// TwinCAT 3 PLC project HeatPumpTestBenchControl
// ProgramVersion: 3.1.4022.1
// CompilerDefines: VISU_USEPROPERTYINFO
// libraries:
//   Tc2_ControllerToolbox, * (Beckhoff Automation GmbH)
//   Tc2_Standard, * (Beckhoff Automation GmbH)
//   Tc2_System, * (Beckhoff Automation GmbH)
//   Tc2_TempController, * (Beckhoff Automation GmbH)
//   Tc2_Utilities, * (Beckhoff Automation GmbH)
//   Tc3_Module, * (Beckhoff Automation GmbH)
//   VisuDialogs, * (System)
// project tree:
//   DUTs/ E_PowMeas.TcDUT (not stored), E_Press.TcDUT (not stored), E_TempSensVR10.TcDUT (not stored), E_TempSensPT100.TcDUT (not stored), E_IndexPowMeas.TcDUT (not stored), E_SMStatus.TcDUT (not stored), E_TempSensVR11.TcDUT (not stored), E_Terminals.TcDUT (not stored), ST_InputVar.TcDUT (not stored), ST_InputVar_PowMeas.TcDUT (not stored), ST_OutputVar.TcDUT (not stored), ST_PumpTime.TcDUT (not stored)
//   / GlobalTextList.TcGTLO (not stored), PlcTask.TcTTO (not stored), Visualization Manager.TcVMO (not stored)
//   GVLs/ DigOutputs.TcGVL (not stored), HeatingCurve.TcGVL (not stored), AnaOutputs.TcGVL (not stored), PID.TcGVL (not stored), PowMeas.TcGVL (not stored), Pressures.TcGVL (not stored), PumpTiming.TcGVL (not stored), StateMachine.TcGVL (not stored), SysCheck.TcGVL (not stored), SysCheckParams.TcGVL (not stored), TempConvDat.TcGVL (not stored), Temperatures.TcGVL (not stored), TempSetpoints.TcGVL (not stored), TerminalErrorRT.TcGVL (not stored), TimeProgs.TcGVL (not stored)
//   POUs/ CheckDivDInt.TcPOU (not stored), CheckDivLInt.TcPOU (not stored), CheckDivLReal.TcPOU (not stored), CheckDivReal.TcPOU (not stored), FB_FanControl.TcPOU, MAIN.TcPOU (not stored), P_GetTime.TcPOU (not stored)
//   POUs/Control/ FB_AuxHeatCont.TcPOU (not stored), FB_CyclingControl.TcPOU (not stored), P_ControlMain.TcPOU (not stored)
//   POUs/Control/TemperatureControl/ FB_PIDSuppTemp.TcPOU (not stored), FB_SimpleTempCont.TcPOU (not stored), F_GetTempSP.TcPOU (not stored), I_TempController.TcIO (not stored), P_SHSuppTempPID.TcPOU (not stored)
//   POUs/ErrorHandling/ F_WriteErrLog.TcPOU (not stored), P_EmShutdownAll.TcPOU (not stored), P_EmShutdownBPumpRun.TcPOU (not stored), P_EmShutdownHCPumpRun.TcPOU (not stored), P_EmShutdownPumpsRun.TcPOU (not stored), P_EmShutdownMain.TcPOU (not stored), P_ErrorHandlingMain.TcPOU (not stored), P_WriteErrLog.TcPOU (not stored)
//   POUs/Initialize/ FB_InitPumpTimes.TcPOU (not stored), FB_ReadHeatCurve.TcPOU (not stored), FB_ReadNightMode.TcPOU (not stored), FB_ReadPressTab.TcPOU (not stored), FB_ReadPT100Tab.TcPOU (not stored), FB_ReadTempResTabVR11.TcPOU (not stored), P_InitMain.TcPOU (not stored), FB_ReadTempResTabVR10.TcPOU (not stored), FB_InitTimes.TcPOU (not stored)
//   POUs/Read/ F_LinSens.TcPOU (not stored), F_NTCSens.TcPOU (not stored), F_PowMeasPhase.TcPOU (not stored), P_PowMeas.TcPOU (not stored), P_ReadMain.TcPOU (not stored), P_TestVals.TcPOU (not stored)
//   POUs/SystemCheck/ F_CheckAmbTemp.TcPOU (not stored), F_CheckBrinePressure.TcPOU (not stored), F_CheckCompCycPress.TcPOU (not stored), F_CheckCompOutTemp.TcPOU (not stored), F_CheckHeatCirPress.TcPOU (not stored), F_CheckHeatCirTemp.TcPOU (not stored), F_CheckPhaseSeq.TcPOU (not stored), F_CheckSens.TcPOU (not stored), F_CheckTerm.TcPOU (not stored), P_SysCheckMain.TcPOU (not stored)
//   POUs/Write/ F_ConvLinAnaOutp.TcPOU (not stored), F_PumpConvPercVolt.TcPOU (not stored), FB_RampPump.TcPOU (not stored), P_WriteMain.TcPOU (not stored)
//   VISUs/ Vis_ManCont.TcVIS (not stored), StandardVis.TcVIS (not stored)
// real-time tasks:
//   TASK PlcTask: cycle T#10ms, priority 20, ADS port 350
// I/O:
//   DEVICE Device 1 (EtherCAT) (disabled), AmsNetId 134.61.132.51.2.1
//     Coupler (EK1100) [EK1100 EtherCAT Coupler (2A E-Bus)]
//       InpPressSens (EL3064) [EL3064 4Ch. Ana. Input 0-10V]
//       InpTempSens1 (EL3204-0200) [EL3204-0200 4Ch. Ana. In. PT1000 (RTD)]
//       InpTempSens2 (EL3204-0200) [EL3204-0200 4Ch. Ana. In. PT1000 (RTD)]
//       InpTempSens3 (EL3204-0200) [EL3204-0200 4Ch. Ana. In. PT1000 (RTD)]
//       InpPowMeas (EL3403-0010) [EL3403-0010 3Ch. Power Measuring, 5A]
//       AnalogOutp (EL4004) [EL4004 4Ch. Ana. Output 0-10V, 12bit]
//       OutpSwitchValv (EL2652) [EL2652 2Ch. Relay Output, CO (230V AC / 30V DC)]
//       OutpCont (EL2622) [EL2622 2Ch. Relay Output, NO (230V AC / 30V DC)]
//       InpTempSens3wire (EL3214) [EL3214 4Ch. Ana. Input PT100 (RTD)]

// ---- POUs/FB_FanControl.TcPOU
FUNCTION_BLOCK FB_FanControl
VAR_INPUT
	fSpeed	:	REAL;		//Fan speed setpoint 0..100%
END_VAR
VAR
	fSpeedSetRaw  AT%Q*	: INT 	:=0; 	//Raw value for terminal => send to valve
END_VAR
VAR CONSTANT
		fFactor : REAL :=327.67;	// factor for calculating the terminal integer values (from percentage to int)
END_VAR

fSpeedSetRaw := REAL_TO_INT(fSpeed*fFactor);

END_FUNCTION_BLOCK
